TYPE ST_BowlFeeder :
	STRUCT
		bOut_Vibrate			AT%Q*	: BOOL;
		bOut_BlowAlign			AT%Q*	: BOOL;
		bIn_NoMaterial			AT%I*	: BOOL;
		bIn_LowLevelMaterial	AT%I*	: BOOL;
		bIn_UnitInPosition		AT%I*	: BOOL;
	END_STRUCT
END_TYPE

(* stored: Version 1.1.0.1, ProductVersion 3.1.4024.12
   DUT ST_BowlFeeder: Id {2416d31b-1a31-4a5e-9593-0772e50d6712} *)
